// Delta ASDA-A2 servo
FUNCTION_BLOCK Fb_DevAxisDelta EXTENDS Fb_DevAxis
VAR
	// Parameters 
		stMParMaxAcc : Udt_Parameter := (fMaximum := 999999, fMinimum := 0, fValue := 0)	; // Parameter for maximum acceleration
		stMParMaxDec : Udt_Parameter := (fMaximum := 999999, fMinimum := 0, fValue := 0)	; // Parameter for maximum Deceleration
		stMparMaxVelo: Udt_Parameter := (fMaximum := 999999, fMinimum := 0, fValue := 0)	; // Parameter for maximum velocity

		
	bResetCalibrationFlag : BOOL := TRUE; // When TRUE, the calibration bit (homing OK) will be reset. Set to TRUE on homing faults.
	fbHomeResetCalibrationFlag:MC_Home;
END_VAR

SUPER^();

fbHomeResetCalibrationFlag(
  Execute:=bResetCalibrationFlag,
  HomingMode:=MC_ResetCalibration,
  Axis:=AxisRef
);
bResetCalibrationFlag R= fbHomeResetCalibrationFlag.Done;

IF bHomed AND (NOT AxisRef.NcToPlc.StateDWord.1) THEN
	bHomed := FALSE;
	bError					:= TRUE							;
	stFault.Active 			:= TRUE 						;
	stFault.Description		:= 'Axis no longer homed';
	stFault.FaultType		:= E_FaultTypes.FF				;	
END_IF

METHOD PUBLIC CmdHome : BOOL
VAR_INPUT
	fPosition 		: LREAL := 0 ; // Homing position
END_VAR
// set blocked command if halt is active 
bBlockedCommand := fbMcHalt.Active ;

// Enable drive 
bExec_Home 		:= NOT bResetCalibrationFlag; 
bInternalEnable	:= TRUE ;

// copy parameters
fbMcHome.Position 	:= fPosition 	;

// Set feedback output
CmdHome := fbMcHome.Done ;
END_METHOD

METHOD PUBLIC CmdMoveAbs : BOOL
VAR_INPUT
	fPosition	:	LREAL 	; // target position
	fVelocity	: 	LREAL 	; // Maximum velocity [units/sec]
	mcBuffermode: 	MC_BufferMode ; // Buffermode defines how the previous command is executed.
END_VAR
VAR
	bNewCommandReceived : BOOL ;
END_VAR
IF (NOT AxisRef.NcToPlc.StateDWord.1) THEN
	bError					:= TRUE							;
	stFault.Active 			:= TRUE 						;
	stFault.Description		:= 'Unable to execute move command, axis not homed';
	stFault.FaultType		:= E_FaultTypes.FF				;	
ELSE
	CmdMoveAbs := SUPER^.CmdMoveAbs(fPosition := fPosition, fVelocity := fVelocity, mcBuffermode := mcBuffermode);
END_IF
END_METHOD

METHOD INTERNAL ExecHome : BOOL
VAR_INPUT
END_VAR
SUPER^.ExecHome();

bResetCalibrationFlag S= fbMcHome.Error;
END_METHOD

METHOD INTERNAL ExecReset : BOOL
IF AxisRef.Status.Coupled THEN 
	bResetDone 	:= NOT AxisRef.Status.Error;
	bExec_Reset	R= bResetDone  ;
	RETURN;
END_IF

// ===== reset command =====
	bError 		:= AxisRef.Status.Error OR AxisRef.Status.DriveDeviceError; 
	bExec_Reset	R= fbMcReset.Done  ;

// ==== execute reset functions =====
fbMcReset	( 	Execute	:= bExec_Reset,
				Axis	:= AxisRef ); 
				
// ===== Set feedback =====
	bResetDone 	S= fbMcReset.Done  ;
	bResetDone	R= AxisRef.Status.Error ;
	tonResetDone (IN	:= bResetDone);

// ===== reset limitations =====
	bCmdSafeSpeed 	:= FALSE ;

	
// Reset fault handling 
	IF fbMcReset.Error THEN 
		bError					:= TRUE							;
		stFault.Active 			:= TRUE 						;
		stFault.Description		:= CONCAT('Reset Fault ', UDINT_TO_STRING(fbMcReset.ErrorID));
		stFault.FaultType		:= E_FaultTypes.FF				;
	END_IF
END_METHOD

METHOD PUBLIC Init : BOOL
VAR_INPUT
	// Message location data
	nId			: UINT ; // Identification number of object
	nParentId	: UDINT ; // Id of higher level If aplicable (0 = no parent)
	
	// Config Bits
	bIcfCmdVelocityRpm	: BOOL := FALSE ; // input speeds in Rpm
	bIcfEnableForward 	: BOOL := TRUE 	; // Enable forward motion
	bIcfEnableReverse	: BOOL := TRUE 	; // Enable reverse motion
	bIcfAlwaysEnable	: BOOL := FALSE ; // 1 = Axis always enabled, 0 = Axis disabled at Idle 
	bIcfModuloAxis		: BOOL := FALSE ; // Show axis position as modulo
	bIcfSTOPresent		: BOOL := FALSE ; // Axis safe torque off is present
	bIcfNCHomeSensor	: BOOL := FALSE ; // Homing sensor is inverted (NC)	
	// Config Values 
	mcHomingMode 		: MC_HomingMode := MC_HomingMode.MC_DefaultHoming; 
	fHomePosition		: LREAL := 0 	; // set position at homing
	fSafeOverride		: LREAL := 10	; // Safe velocity override [%]
	nEncTurnoverVal 	: LREAL := 360	; // encoder turnover value 
	tEnableDelay		: time 	:= T#0MS; // Time between axis enable command and motion command execution (0 := no delay active)	
	tDisabledelay		: TIME 	:= T#100MS; // Axis idle time before axis is disabled 
END_VAR
// ====== Calculate device id =====
	bInitOk :=	ExecIdentifyDevice(nId,nParentId, E_ComponentTypes.Axis) AND bInitOk;

// ====== Set manual device type ======
	eDevType := E_Devices.Axis ;	
	
// ===== Write parameters =====
	stMParMaxAcc.nNumber		:= stIdentity.nLocationId + 1;
	stMParMaxAcc.sDiscription 	:= CONCAT(STR1 := stIdentity.sName, STR2:= ' hardware maximum acceleration (0 = HWMaximum)'); 
	stMParMaxAcc.sName			:= CONCAT(STR1 := stIdentity.sName, STR2:= 'Hard max acceleration');
	stMParMaxAcc.sType			:= 'MPar';
	stMParMaxAcc.sUnit			:= 'unit/s^2';
	
	stMParMaxDec.nNumber		:= stIdentity.nLocationId + 2;
	stMParMaxDec.sDiscription 	:= CONCAT(STR1 := stIdentity.sName, STR2:= ' hardware maximum deceleration (0 = HWMaximum)'); 
	stMParMaxDec.sName			:= CONCAT(STR1 := stIdentity.sName, STR2:= 'Hard max deceleration');
	stMParMaxDec.sType			:= 'MPar';
	stMParMaxDec.sUnit			:= 'unit/s^2';
	
	stMparMaxVelo.nNumber		:= stIdentity.nLocationId + 3;
	stMparMaxVelo.sDiscription 	:= CONCAT(STR1 := stIdentity.sName, STR2:= ' hardware maximum velocity'); 
	stMparMaxVelo.sName			:= CONCAT(STR1 := stIdentity.sName, STR2:= 'Hard max velocity');
	stMparMaxVelo.sType			:= 'MPar';
	stMparMaxVelo.sUnit			:= 'Units/s';

	refFbParHandler.CmdAddParameter(refParameter := stMParMaxAcc);
	refFbParHandler.CmdAddParameter(refParameter := stMParMaxDec);
	refFbParHandler.CmdAddParameter(refParameter := stMparMaxVelo);

// ===== set axis configuration =====	
	fMaxAcc	:= stMParMaxAcc.fValue;
	fMaxDec	:= stMParMaxDec.fValue;	
	fMaxVelo:= stMparMaxVelo.fValue;

	fCmdAcc 		:= fMaxAcc;
	fCmdDecc		:= fMaxDec;

// ===== Configure Axis =====
	// ***** Config Bits *****
		THIS^.bIcfCmdVelocityRpm	:= bIcfCmdVelocityRpm	; // Enable speed inputs in Rpm
		THIS^.bIcfEnableForward 	:= bIcfEnableForward 	; // Enable forward motion
		THIS^.bIcfEnableReverse		:= bIcfEnableReverse	; // Enable reverse motion
		THIS^.bIcfAlwaysEnable		:= bIcfAlwaysEnable		; // Always enable motor and brake if safety is ok
		THIS^.bIcfModuloAxis		:= bIcfModuloAxis		; // show axis position as modulo
		THIS^.bIcfSTOPresent		:= bIcfSTOPresent		; // Axis has safe torque off function
		THIS^.bIcfNCHomeSensor		:= bIcfNCHomeSensor		; // Axis homing sensor is NC	
	// ***** config homing Mode ***** 
 		THIS^.mcHomingMode 			:= mcHomingMode ; // set homing mode
		THIS^.fHomePosition			:= fHomePosition;
	// ***** Velocity settings *****
		THIS^.fSafeOverride			:= fSafeOverride	; 	
	// ***** Encoder values *****
		THIS^.fEncoderTurnoverValue := nEncTurnoverVal	; // turnover value for encoder = 25.6 mm per rev * 4096 revolutions 
	// ***** Time delay enable off *****
		THIS^.tEnableDelay		:= tEnableDelay	;
		THIS^.tDisableDelay 	:= tDisabledelay ;		
		
// ===== configure parameters =====
	ParAccManualScaling.fMinimum 		:= 1 	;
	ParAccManualScaling.fMaximum		:= 100 	;
	ParAccManualScaling.nNumber 		:= stIdentity.nLocationId + 1;
	ParAccManualScaling.sDiscription  	:= CONCAT( STR1 := stIdentity.sName, STR2 := ' percentage of acceleration used for jogging');
	ParAccManualScaling.sName			:= CONCAT( STR1 := stIdentity.sName, STR2 := 'Manual acc scaling');
	ParAccManualScaling.sType			:= 'Mpar';
	ParAccManualScaling.sUnit			:= '%';
	refFbParHandler.CmdAddParameter( refParameter := ParAccManualScaling );

	
	ParDecManualScaling.fMinimum 		:= 1 	;
	ParDecManualScaling.fMaximum		:= 100 	;
	ParDecManualScaling.nNumber 		:= stIdentity.nLocationId + 2;
	ParDecManualScaling.sDiscription  	:= CONCAT( STR1 := stIdentity.sName, STR2 := ' percentage of deceleration used for jogging');
	ParDecManualScaling.sName			:= CONCAT( STR1 := stIdentity.sName, STR2 := 'Manual dec scaling');
	ParDecManualScaling.sType			:= 'Mpar';
	ParDecManualScaling.sUnit			:= '%';
	refFbParHandler.CmdAddParameter( refParameter := ParAccManualScaling );

// ===== reset axis state indicators ======
	bError 	:= FALSE;

// ====== Set init to done =======
	bInitOk := TRUE;
	Init := bInitOk;
END_METHOD

END_FUNCTION_BLOCK

(* stored: Version 1.1.0.1, ProductVersion 3.1.4024.11
   POU Fb_DevAxisDelta: Id {63a8c96e-3fc0-001c-2116-24486a7558ba}, SpecialFunc None
   Folder Command Methods: Id {6ff04a08-145f-0075-3081-8a253c264400}
   Folder Private: Id {411a3c08-0cd0-0279-3d64-90e3acd48f7f}
   Folder Motion: Id {6c2d68a6-87c9-02f7-38fa-57b088d1fb56}
   Folder Organization: Id {3dbff440-0f61-0a96-00dd-248ac60e3867}
   Method CmdHome: Id {c659379d-7a9a-0709-3350-5e8b08b834ec}
   Method CmdMoveAbs: Id {a54c6e1a-38da-0009-0a84-54aa7056f5c4}
   Method ExecHome: Id {46e109e7-8a56-0014-319d-132073728766}
   Method ExecReset: Id {2608dc0b-c27b-03ab-2a5f-162cf169c209}
   Method Init: Id {2b37d305-8771-08f4-26c5-28ec9072ede6} *)
